FUNCTION_BLOCK FB_ADS_DVTSHEETALIGNMENT EXTENDS FB_AdsBlockBase
VAR
  // ---------------------------------
  // ADS interface block specific
  sO_Message         : ST_ADS_MSG_IF;
  
  bI_Enable          : BOOL := TRUE;    (*Enable processing*)

  bI_UsePrintMark    : BOOL := TRUE;    (*Enable processing of print marks*)
  sI_PrintMarkSizeX  : ST_VAR_IN_REAL;  (*Print mark X size [mm]*)
  sI_PrintMarkSizeY  : ST_VAR_IN_REAL;  (*Print mark Y size [mm]*)

  sI_HeadGap         : ST_VAR_IN_REAL;  (*Gap between head and substrate [mm]*)

  lI_SegmentSize     : UDINT;           (*Distance between two images in pixel*)
  lI_SegmentCount    : UDINT;           (*Number of images*)
  fI_SegmentAngle    : REAL;            (*Angle between two segments in deg*)

  sI_DeltaX          : ST_VAR_IN_REAL;  (*X offset between camera marks [mm]*)

  bI_IsMaintenanceJob: BOOL;            (*Maintenance job: disable shift and rotation*)

  (*Out*)
  sO_CurrentAngle    : ST_VAR_OUT_REAL; (*Last measured angle in deg*)
  lO_CurrentYShift   : UDINT;           (*Last measured Y Shift in Pixel*)

  bO_RangeErrorAngle : BOOL;            (*Measured angle out of range*)
  bO_RangeErrorShift : BOOL;            (*Measured shift out of range*)

  // ---------------------------------
END_VAR
VAR PERSISTENT
  aR_Pattern         : UDINT;           (*check pattern for rem validity*)
  bR_Enable          : BOOL;            (*remanent: *)
  bR_UsePrintMark    : BOOL;            (*remanent: *)
  fR_PrintMarkSize_X : REAL;            (*remanent: *)
  fR_PrintMarkSize_Y : REAL;            (*remanent: *)
  fR_HeadGap         : REAL;            (*remanent: head gap in [mm]*)
  fR_DeltaX          : REAL;            (*remanent: *)
END_VAR

PROPERTY bEnable : BOOL
GET
bEnable   := bI_Enable;   // Set ads interface variable
bR_Enable := bI_Enable;   // Update remanent variable
END_GET
SET
bI_Enable := bEnable;   // set interface variable
bR_Enable := bEnable;   // update remanent variable
END_SET
END_PROPERTY

PROPERTY bIsMaintenanceJob : BOOL
GET
bIsMaintenanceJob := bI_IsMaintenanceJob;   // Set ads interface variable
END_GET
SET
bI_IsMaintenanceJob := bIsMaintenanceJob;   // Set ads interface variable
END_SET
END_PROPERTY

PROPERTY bRangeErrorAngle : BOOL
SET
bO_RangeErrorAngle := bRangeErrorAngle;
END_SET
END_PROPERTY

PROPERTY bRangeErrorShift : BOOL
SET
bO_RangeErrorShift := bRangeErrorShift;
END_SET
END_PROPERTY

PROPERTY bUsePrintMark : BOOL
GET
bUsePrintMark   := bI_UsePrintMark;   // Set ads interface variable
bR_UsePrintMark := bI_UsePrintMark;   // Update remanent variable
END_GET
SET
bI_UsePrintMark := bUsePrintMark;   // set interface variable
bR_UsePrintMark := bUsePrintMark;   // update remanent variable
END_SET
END_PROPERTY

METHOD config
VAR_INPUT
  bPrintMarkSizeX_Exist : BOOL;
  aPrintMarkSizeX_Unit  : STRING;
  fPrintMarkSizeX_Min   : REAL;
  fPrintMarkSizeX_Max   : REAL;
  
  bPrintMarkSizeY_Exist : BOOL;
  aPrintMarkSizeY_Unit  : STRING;
  fPrintMarkSizeY_Min   : REAL;
  fPrintMarkSizeY_Max   : REAL;
  
  bHeadGap_Exist        : BOOL;
  aHeadGap_Unit         : STRING;
  fHeadGap_Min          : REAL;
  fHeadGap_Max          : REAL;

  bDeltaX_Exist         : BOOL;
  aDeltaX_Unit          : STRING;
  fDeltaX_Min           : REAL;
  fDeltaX_Max           : REAL;
  
  bCurrentAngle_Exist   : BOOL;
  aCurrentAngle_Unit    : STRING;
  fCurrentAngle_Min     : REAL;
  fCurrentAngle_Max     : REAL;
END_VAR
sI_PrintMarkSizeX.bC_Exist := bPrintMarkSizeX_Exist;
sI_PrintMarkSizeX.aC_Unit  := aPrintMarkSizeX_Unit;
sI_PrintMarkSizeX.fC_Min   := fPrintMarkSizeX_Min;
sI_PrintMarkSizeX.fC_Max   := fPrintMarkSizeX_Max;
sI_PrintMarkSizeY.bC_Exist := bPrintMarkSizeY_Exist;
sI_PrintMarkSizeY.aC_Unit  := aPrintMarkSizeY_Unit;
sI_PrintMarkSizeY.fC_Min   := fPrintMarkSizeY_Min;
sI_PrintMarkSizeY.fC_Max   := fPrintMarkSizeY_Max;
sI_HeadGap.bC_Exist        := bHeadGap_Exist;
sI_HeadGap.aC_Unit         := aHeadGap_Unit;
sI_HeadGap.fC_Min          := fHeadGap_Min;
sI_HeadGap.fC_Max          := fHeadGap_Max;
sI_DeltaX.bC_Exist         := bDeltaX_Exist;
sI_DeltaX.aC_Unit          := aDeltaX_Unit;
sI_DeltaX.fC_Min           := fDeltaX_Min;
sI_DeltaX.fC_Max           := fDeltaX_Max;
sO_CurrentAngle.bC_Exist   := bCurrentAngle_Exist;
sO_CurrentAngle.aC_Unit    := aCurrentAngle_Unit;
sO_CurrentAngle.fC_Min     := fCurrentAngle_Min;
sO_CurrentAngle.fC_Max     := fCurrentAngle_Max;

sO_CurrentAngle.bC_Exist   := FALSE;

initRemVar();
END_METHOD

PROPERTY fDeltaX : REAL
GET
fDeltaX   := sI_DeltaX.fI_Val;   // Set ads interface variable
fR_DeltaX := sI_DeltaX.fI_Val;
END_GET
END_PROPERTY

// HeadGap in [mm]
PROPERTY fHeadGap : LREAL
GET
fHeadGap   := sI_HeadGap.fI_Val;   // Set ads interface variable
fR_HeadGap := sI_HeadGap.fI_Val;   // Update remanent variable
END_GET
SET
sI_HeadGap.fI_Val := TO_REAL(fHeadGap);   // set interface variable
fR_HeadGap        := TO_REAL(fHeadGap);   // update remanent variable
END_SET
END_PROPERTY

PROPERTY fMarkSizeX : REAL
GET
fMarkSizeX         := sI_PrintMarkSizeX.fI_Val;   // Set ads interface variable
fR_PrintMarkSize_X := sI_PrintMarkSizeX.fI_Val;   // Update remanent variable
END_GET
END_PROPERTY

PROPERTY fMarkSizeY : REAL
GET
fMarkSizeY         := sI_PrintMarkSizeY.fI_Val;   // Set ads interface variable
fR_PrintMarkSize_Y := sI_PrintMarkSizeY.fI_Val;   // Update remanent variable
END_GET
END_PROPERTY

PROPERTY fO_CurrentAngle : LREAL
SET
sO_CurrentAngle.fO_Val := tO_REAL(fO_CurrentAngle);
END_SET
END_PROPERTY

PROPERTY fSegmentAngle : REAL
GET
fSegmentAngle := fI_SegmentAngle;   // Set ads interface variable
END_GET
END_PROPERTY

METHOD PROTECTED initRemVar
(*load default initial values if pattern was invalid*)
IF aR_Pattern <> 16#ABCD THEN
  aR_Pattern  := 16#ABCD;  
  bR_Enable   := TRUE;
  bR_UsePrintMark := 0;
  fR_PrintMarkSize_X := 0;
  fR_PrintMarkSize_Y := 0;
  fR_HeadGap  := 2;
  fR_DeltaX := 0;
END_IF

bI_Enable := bR_Enable;
bI_UsePrintMark := bR_UsePrintMark;
sI_PrintMarkSizeX.fI_Val := fR_PrintMarkSize_X;
sI_PrintMarkSizeY.fI_Val := fR_PrintMarkSize_Y;
sI_HeadGap.fI_Val := fR_HeadGap;
sI_DeltaX.fI_Val := fR_DeltaX;
END_METHOD

PROPERTY nO_CurrentYShift : UDINT
SET
lO_CurrentYShift := nO_CurrentYShift;
END_SET
END_PROPERTY

PROPERTY nSegmentCount : UDINT
GET
nSegmentCount := lI_SegmentCount;   // Set ads interface variable
END_GET
END_PROPERTY

PROPERTY nSegmentSize : UDINT
GET
nSegmentSize := lI_SegmentSize;   // Set ads interface variable
END_GET
END_PROPERTY

(*
  Setup constant ADS Block definitions.
  HOWTO: in abstract implmentation call
      init(aVersion:=, aType:=, nType:=, eLayer:=);
*)
METHOD  setup
init(aVersion:='01.00.10', aType:='DvtSheetAlignment', nType:=ePr_BLK_SA, eLayer:=E_AdsLayer.Structural);
END_METHOD

PROPERTY sMsgInterface : POINTER TO ST_ADS_MSG_IF
GET
sMsgInterface := ADR(sO_Message);
END_GET
END_PROPERTY

END_FUNCTION_BLOCK

(* stored: Version 1.1.0.1, ProductVersion 3.1.4024.11
   POU FB_ADS_DVTSHEETALIGNMENT: Id {767ea748-f391-4f32-9fdd-aa405f60b0a7}, SpecialFunc None
   Folder Ads: Id {298afe55-d105-4068-a77b-7734006dad5e}
   Property bEnable: Id {9450c399-c0da-463f-8664-2aded51fccca}
   Get Get: Id {d5ca6d74-a4e3-49e2-9cd3-b2221ff4dd82}
   Set Set: Id {e32895c2-f853-47bc-b719-07c9c7e44508}
   Property bIsMaintenanceJob: Id {78601085-31dc-476e-9363-45a2f4f544ec}
   Get Get: Id {813f1b74-992a-4167-8f1d-3fa8314069c4}
   Set Set: Id {ce9d9303-9377-4a95-88c5-e7c45c236367}
   Property bRangeErrorAngle: Id {9097c5f9-4aaa-4522-9f98-4cf174df6d3e}
   Set Set: Id {7d56cfec-891f-4e37-a4cb-5b16c7c25c7d}
   Property bRangeErrorShift: Id {098fa57a-4512-4eb7-b06b-92fce8602911}
   Set Set: Id {664dcf62-fa37-4b61-848c-c60ff901974d}
   Property bUsePrintMark: Id {b9565c86-8818-46e9-82b5-08357c08c60b}
   Get Get: Id {bf3af2db-46fd-4d34-b128-89617ec23634}
   Set Set: Id {d6af134e-8079-4689-b9e7-4800e1e2e8ef}
   Method config: Id {310c53a1-bb03-42bc-8be5-9521b96a931e}
   Property fDeltaX: Id {cc2c3a05-6041-427e-bc96-aaff9df29975}
   Get Get: Id {5311e5a7-89b7-4895-9ebf-7d2daea3e531}
   Property fHeadGap: Id {e8a54815-d0df-4e0c-900f-5afd2ec6c964}
   Get Get: Id {5e61d2ef-dd66-4d21-8268-de3a94d9ae2f}
   Set Set: Id {ff2b860b-9bde-41cd-bbc9-ba2a96f007b3}
   Property fMarkSizeX: Id {11e9f71d-bd48-4f5c-a55c-d6c22678be31}
   Get Get: Id {9a187e7b-b4f1-466e-bb14-132ec9c48cd8}
   Property fMarkSizeY: Id {77596c7f-5509-4b50-b650-6f285d00aee6}
   Get Get: Id {f9e7a072-d3f1-48d8-8ede-4be6915325c4}
   Property fO_CurrentAngle: Id {06f18c7c-e634-483d-ace3-7982e879b6ba}
   Set Set: Id {befcecb7-6770-45a6-8073-e06ce493ff7b}
   Property fSegmentAngle: Id {6ff6dcb2-1300-4275-aab3-407a4825a282}
   Get Get: Id {cc15a034-12b1-48ce-8450-9942dd4ab675}
   Method initRemVar: Id {a397f808-fb60-4152-b71a-46f5708a7161}
   Property nO_CurrentYShift: Id {b4a6da06-f36a-40f8-a531-162fe31d94de}
   Set Set: Id {401c5b63-184a-46de-9d43-e502627f11b1}
   Property nSegmentCount: Id {5a3c98a2-4c14-4585-9e8c-1bff18f71632}
   Get Get: Id {0def26bd-50c5-4bee-a092-9299d20f14d9}
   Property nSegmentSize: Id {75eedc24-9be1-47a3-8b12-44901a98b7ef}
   Get Get: Id {c2f16be4-d134-41bc-baaf-1bc0997893eb}
   Method setup: Id {ae53dba6-3a79-468e-88f6-50b94b8da441}
   Property sMsgInterface: Id {3007b5f4-968d-44ed-a66b-c0ffb62b246d}
   Get Get: Id {4e5925a9-bdb0-4bf9-8e26-de5a5ded8c3b} *)
